FUNCTION_BLOCK FB_Component_DualValve IMPLEMENTS I_Component
VAR_INPUT
// Interface vars
	sName			: STRING[20];
	bEnable     	: BOOL;
	//eMode       	: E_ComponentMode;
END_VAR

VAR_IN_OUT
	bOutputA		: BOOL;
	bOutputB		: BOOL;
END_VAR

VAR_OUTPUT
	// interface vars
	eState			: E_ComponentState;
	iErrorCode		: INT;
	sStatusText 	: STRING[50];
END_VAR

METHOD M_Extend : BOOL
VAR_INPUT
END_VAR
IF bEnable AND eState = E_ComponentState.READY THEN
	bOutputA := TRUE;
	bOutputB := FALSE;	
END_IF;
END_METHOD

{warning 'add method implementation '}
METHOD M_Halt : BOOL
bOutputA := FALSE;
bOutputB := FALSE;
eState := E_ComponentState.HALTED;
END_METHOD

METHOD M_Hold : BOOL
VAR_INPUT
END_VAR
IF bEnable AND eState = E_ComponentState.READY THEN
	bOutputA := FALSE;
	bOutputB := FALSE;	
END_IF;
END_METHOD

METHOD M_Retract : BOOL
VAR_INPUT
END_VAR
IF bEnable AND eState = E_ComponentState.READY THEN
	bOutputA := FALSE;
	bOutputB := TRUE;	
END_IF;
END_METHOD

{warning 'add method implementation '}
METHOD M_Start : BOOL
IF eState <> E_ComponentState.BUSY THEN
	eState := E_ComponentState.READY;
END_IF;
END_METHOD

{warning 'add method implementation '}
METHOD M_Stop : BOOL
IF eState <> E_ComponentState.BUSY THEN
	eState := E_ComponentState.DONE;
END_IF
END_METHOD

END_FUNCTION_BLOCK

(* stored: Version 1.1.0.1, ProductVersion 3.1.4024.15
   POU FB_Component_DualValve: Id {04d6caaa-12ea-4ca7-b40e-e6e2c47167ec}, SpecialFunc None
   Method M_Extend: Id {7e03a1a2-3117-478d-bc9e-fe754014a4c0}
   Method M_Halt: Id {7e26450e-626a-49e3-bf77-f7d108f47e28}
   Method M_Hold: Id {7bb88dd3-8cd3-406c-a05b-4f33c160f309}
   Method M_Retract: Id {b72d4012-63c2-4591-aa84-c9e3b643667f}
   Method M_Start: Id {bba54da0-4844-47de-8d18-e24d357031dd}
   Method M_Stop: Id {c7fdd13c-07aa-4ec7-8f00-225aca00b1d0} *)
